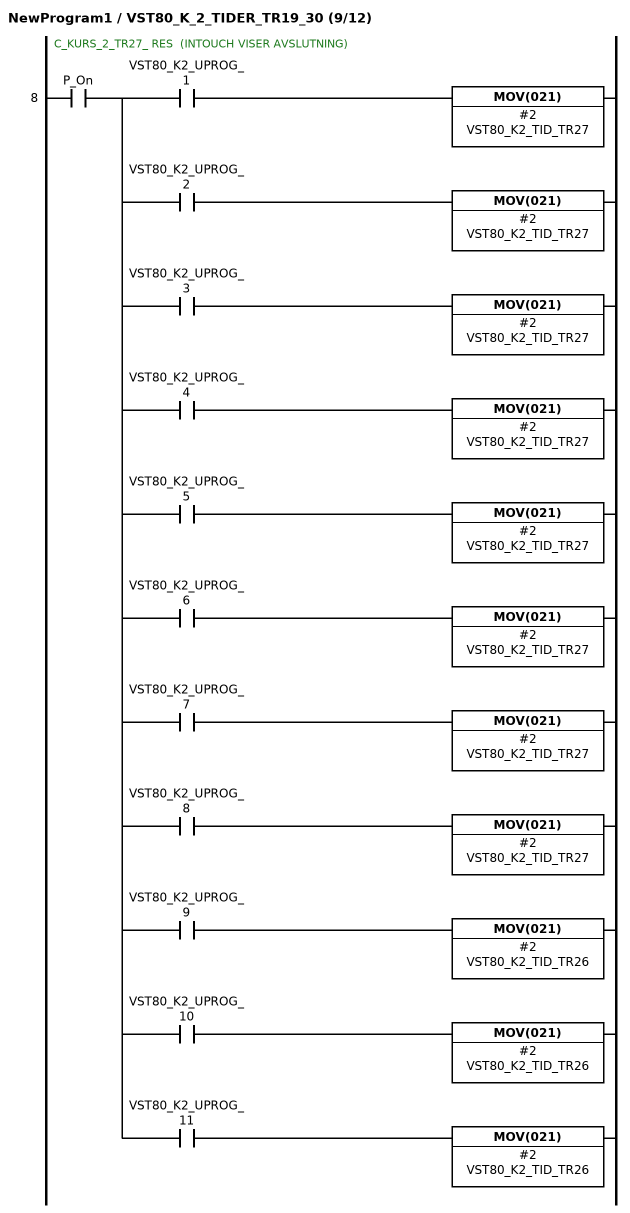
; [picture p192: NewProgram1 / VST80_K_2_TIDER_TR19_30, rungs 8-8]
; rung 8: C_KURS_2_TR27_ RES  (INTOUCH VISER AVSLUTNING)
LD P_On
OUT TR0
AND VST80_K2_UPROG_1
MOV(021) #2 VST80_K2_TID_TR27
LD TR0
AND VST80_K2_UPROG_2
MOV(021) #2 VST80_K2_TID_TR27
LD TR0
AND VST80_K2_UPROG_3
MOV(021) #2 VST80_K2_TID_TR27
LD TR0
AND VST80_K2_UPROG_4
MOV(021) #2 VST80_K2_TID_TR27
LD TR0
AND VST80_K2_UPROG_5
MOV(021) #2 VST80_K2_TID_TR27
LD TR0
AND VST80_K2_UPROG_6
MOV(021) #2 VST80_K2_TID_TR27
LD TR0
AND VST80_K2_UPROG_7
MOV(021) #2 VST80_K2_TID_TR27
LD TR0
AND VST80_K2_UPROG_8
MOV(021) #2 VST80_K2_TID_TR27
LD TR0
AND VST80_K2_UPROG_9
MOV(021) #2 VST80_K2_TID_TR26
LD TR0
AND VST80_K2_UPROG_10
MOV(021) #2 VST80_K2_TID_TR26
LD TR0
AND VST80_K2_UPROG_11
MOV(021) #2 VST80_K2_TID_TR26

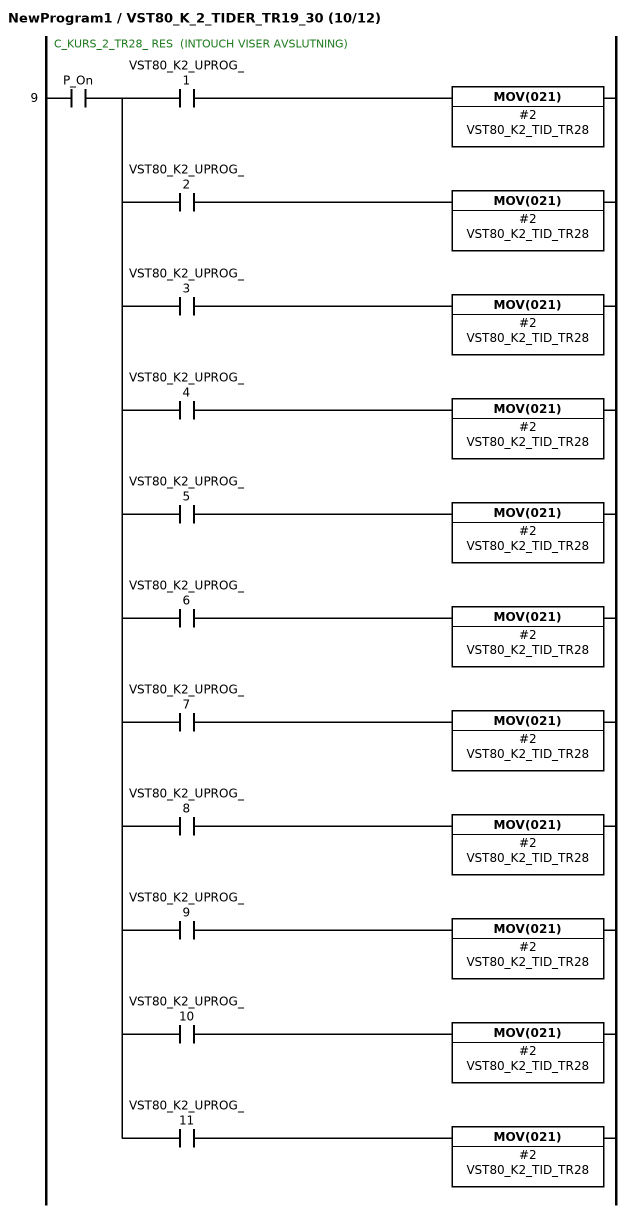
; rung 9: C_KURS_2_TR28_ RES  (INTOUCH VISER AVSLUTNING)
LD P_On
OUT TR0
AND VST80_K2_UPROG_1
MOV(021) #2 VST80_K2_TID_TR28
LD TR0
AND VST80_K2_UPROG_2
MOV(021) #2 VST80_K2_TID_TR28
LD TR0
AND VST80_K2_UPROG_3
MOV(021) #2 VST80_K2_TID_TR28
LD TR0
AND VST80_K2_UPROG_4
MOV(021) #2 VST80_K2_TID_TR28
LD TR0
AND VST80_K2_UPROG_5
MOV(021) #2 VST80_K2_TID_TR28
LD TR0
AND VST80_K2_UPROG_6
MOV(021) #2 VST80_K2_TID_TR28
LD TR0
AND VST80_K2_UPROG_7
MOV(021) #2 VST80_K2_TID_TR28
LD TR0
AND VST80_K2_UPROG_8
MOV(021) #2 VST80_K2_TID_TR28
LD TR0
AND VST80_K2_UPROG_9
MOV(021) #2 VST80_K2_TID_TR28
LD TR0
AND VST80_K2_UPROG_10
MOV(021) #2 VST80_K2_TID_TR28
LD TR0
AND VST80_K2_UPROG_11
MOV(021) #2 VST80_K2_TID_TR28

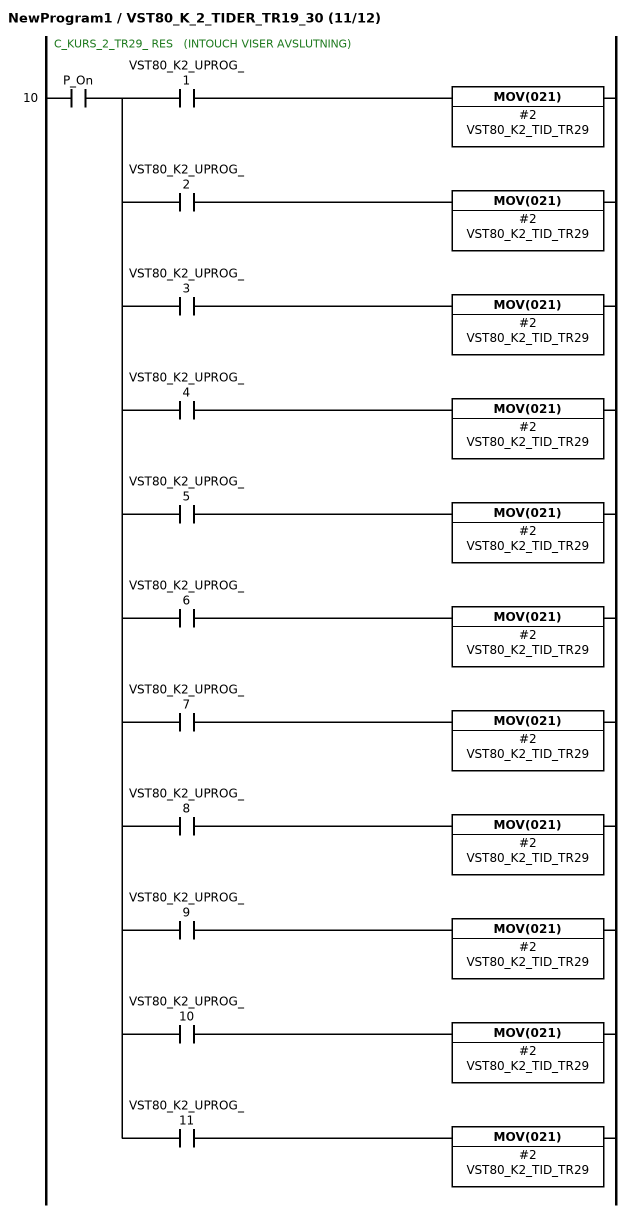
; rung 10: C_KURS_2_TR29_ RES   (INTOUCH VISER AVSLUTNING)
LD P_On
OUT TR0
AND VST80_K2_UPROG_1
MOV(021) #2 VST80_K2_TID_TR29
LD TR0
AND VST80_K2_UPROG_2
MOV(021) #2 VST80_K2_TID_TR29
LD TR0
AND VST80_K2_UPROG_3
MOV(021) #2 VST80_K2_TID_TR29
LD TR0
AND VST80_K2_UPROG_4
MOV(021) #2 VST80_K2_TID_TR29
LD TR0
AND VST80_K2_UPROG_5
MOV(021) #2 VST80_K2_TID_TR29
LD TR0
AND VST80_K2_UPROG_6
MOV(021) #2 VST80_K2_TID_TR29
LD TR0
AND VST80_K2_UPROG_7
MOV(021) #2 VST80_K2_TID_TR29
LD TR0
AND VST80_K2_UPROG_8
MOV(021) #2 VST80_K2_TID_TR29
LD TR0
AND VST80_K2_UPROG_9
MOV(021) #2 VST80_K2_TID_TR29
LD TR0
AND VST80_K2_UPROG_10
MOV(021) #2 VST80_K2_TID_TR29
LD TR0
AND VST80_K2_UPROG_11
MOV(021) #2 VST80_K2_TID_TR29

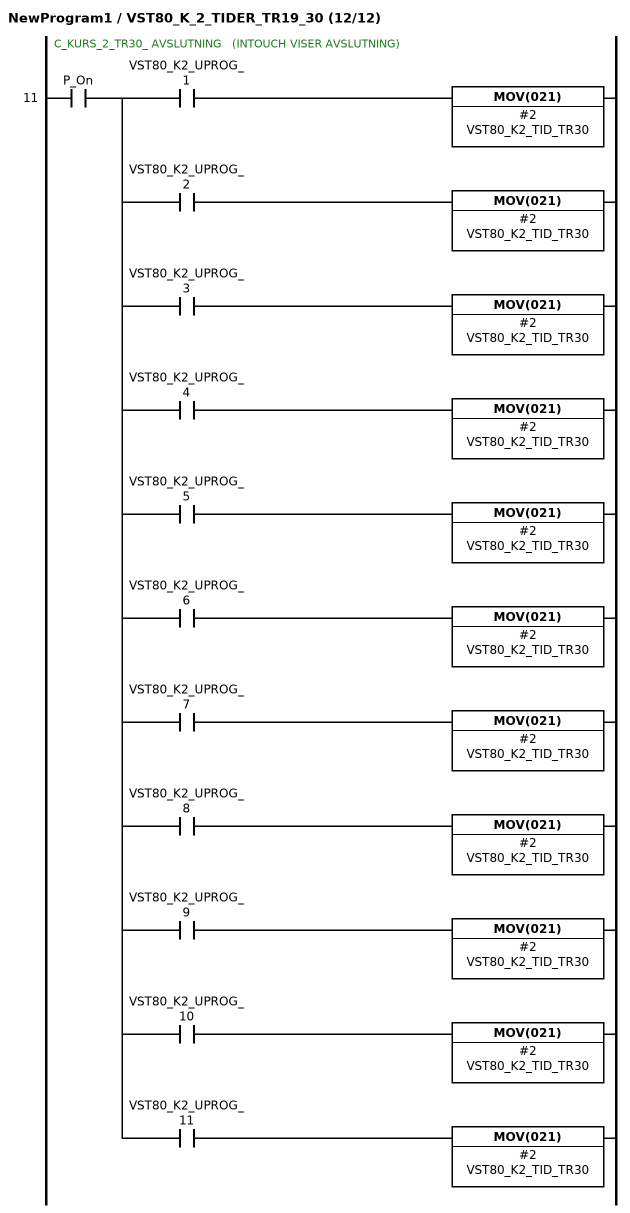
; rung 11: C_KURS_2_TR30_ AVSLUTNING   (INTOUCH VISER AVSLUTNING)
LD P_On
OUT TR0
AND VST80_K2_UPROG_1
MOV(021) #2 VST80_K2_TID_TR30
LD TR0
AND VST80_K2_UPROG_2
MOV(021) #2 VST80_K2_TID_TR30
LD TR0
AND VST80_K2_UPROG_3
MOV(021) #2 VST80_K2_TID_TR30
LD TR0
AND VST80_K2_UPROG_4
MOV(021) #2 VST80_K2_TID_TR30
LD TR0
AND VST80_K2_UPROG_5
MOV(021) #2 VST80_K2_TID_TR30
LD TR0
AND VST80_K2_UPROG_6
MOV(021) #2 VST80_K2_TID_TR30
LD TR0
AND VST80_K2_UPROG_7
MOV(021) #2 VST80_K2_TID_TR30
LD TR0
AND VST80_K2_UPROG_8
MOV(021) #2 VST80_K2_TID_TR30
LD TR0
AND VST80_K2_UPROG_9
MOV(021) #2 VST80_K2_TID_TR30
LD TR0
AND VST80_K2_UPROG_10
MOV(021) #2 VST80_K2_TID_TR30
LD TR0
AND VST80_K2_UPROG_11
MOV(021) #2 VST80_K2_TID_TR30

### Section VST80_K2_TRINN
; Vaskeprogrammet består av 30. hovedtrinn. / Funksjonsbenstabell: 975100-BL48

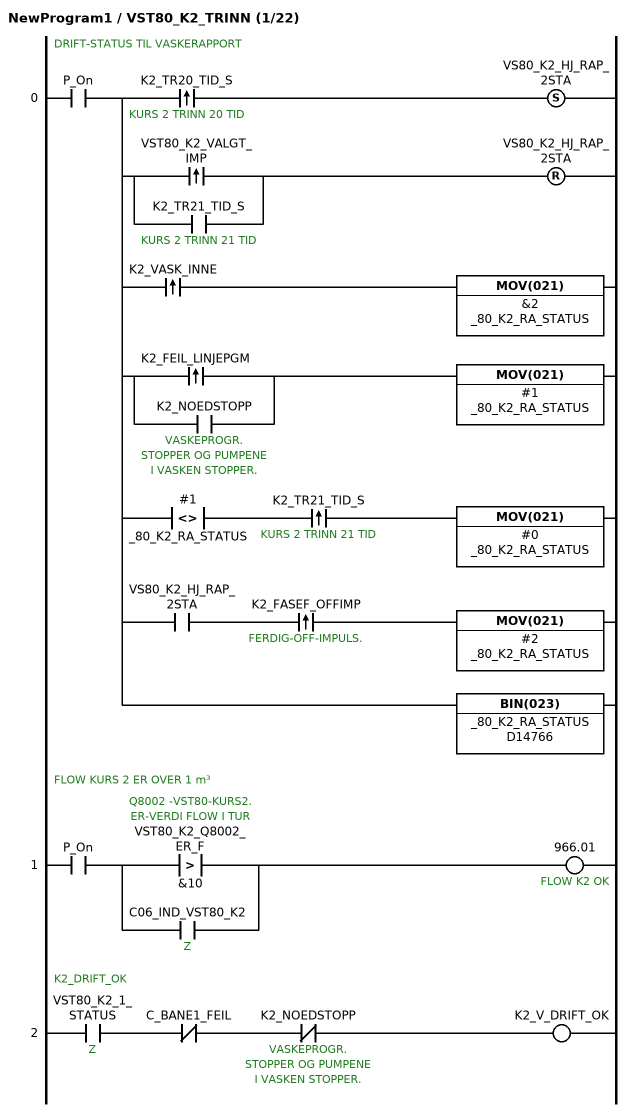
; rung 0: DRIFT-STATUS TIL VASKERAPPORT
LD P_On
OUT TR0
@AND K2_TR20_TID_S  ; KURS 2 TRINN 20 TID
SET VS80_K2_HJ_RAP_2STA
LD TR0
@LD VST80_K2_VALGT_IMP
OR K2_TR21_TID_S  ; KURS 2 TRINN 21 TID
ANDLD
RSET VS80_K2_HJ_RAP_2STA
LD TR0
@AND K2_VASK_INNE
MOV(021) &2 _80_K2_RA_STATUS
LD TR0
@LD K2_FEIL_LINJEPGM
OR K2_NOEDSTOPP  ; VASKEPROGR. STOPPER OG PUMPENE I VASKEN STOPPER.
ANDLD
MOV(021) #1 _80_K2_RA_STATUS
LD TR0
AND<>(305) #1 _80_K2_RA_STATUS
@AND K2_TR21_TID_S  ; KURS 2 TRINN 21 TID
MOV(021) #0 _80_K2_RA_STATUS
LD TR0
AND VS80_K2_HJ_RAP_2STA
@AND K2_FASEF_OFFIMP  ; FERDIG-OFF-IMPULS.
MOV(021) #2 _80_K2_RA_STATUS
LD TR0
BIN(023) _80_K2_RA_STATUS D14766
; rung 1: FLOW KURS 2 ER OVER 1 m³
LD P_On
LD>(320) VST80_K2_Q8002_ER_F &10  ; Q8002 -VST80-KURS2. ER-VERDI FLOW I TUR
OR C06_IND_VST80_K2  ; Z
ANDLD
OUT 966.01  ; FLOW K2 OK
; rung 2: K2_DRIFT_OK
LD VST80_K2_1_STATUS  ; Z
ANDNOT C_BANE1_FEIL
ANDNOT K2_NOEDSTOPP  ; VASKEPROGR. STOPPER OG PUMPENE I VASKEN STOPPER.
OUT K2_V_DRIFT_OK

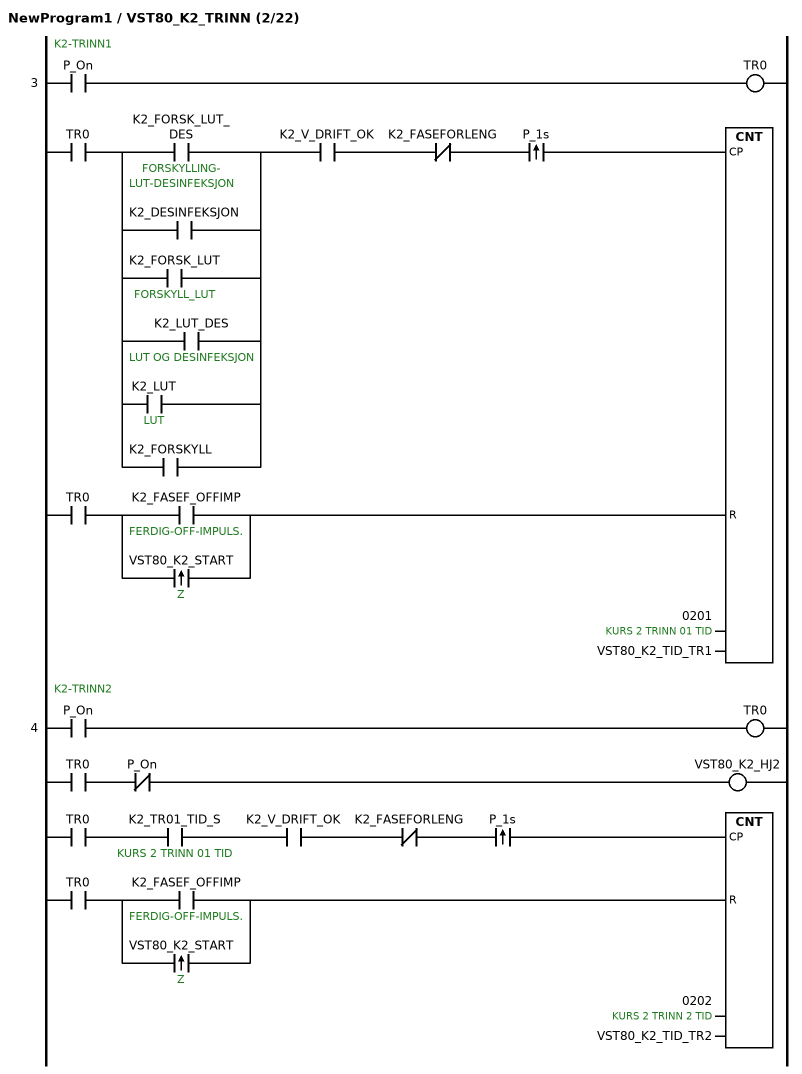
; rung 3: K2-TRINN1
LD P_On
OUT TR0
LD K2_FORSK_LUT_DES  ; FORSKYLLING- LUT-DESINFEKSJON
OR K2_DESINFEKSJON
OR K2_FORSK_LUT  ; FORSKYLL_LUT
OR K2_LUT_DES  ; LUT OG DESINFEKSJON
OR K2_LUT  ; LUT
OR K2_FORSKYLL
ANDLD
AND K2_V_DRIFT_OK
ANDNOT K2_FASEFORLENG
@AND P_1s
LD TR0
LD K2_FASEF_OFFIMP  ; FERDIG-OFF-IMPULS.
@OR VST80_K2_START  ; Z
ANDLD
CNT 0201 VST80_K2_TID_TR1  ; KURS 2 TRINN 01 TID
; rung 4: K2-TRINN2
LD P_On
OUT TR0
ANDNOT P_On
OUT VST80_K2_HJ2
LD TR0
AND K2_TR01_TID_S  ; KURS 2 TRINN 01 TID
AND K2_V_DRIFT_OK
ANDNOT K2_FASEFORLENG
@AND P_1s
LD TR0
LD K2_FASEF_OFFIMP  ; FERDIG-OFF-IMPULS.
@OR VST80_K2_START  ; Z
ANDLD
CNT 0202 VST80_K2_TID_TR2  ; KURS 2 TRINN 2 TID

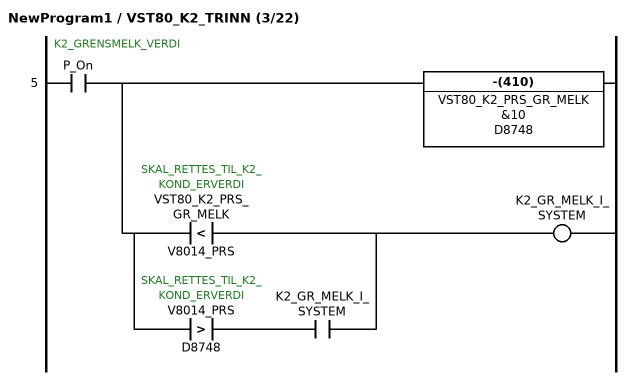
; rung 5: K2_GRENSMELK_VERDI
LD P_On
-(410) VST80_K2_PRS_GR_MELK &10 D8748
LD<(310) VST80_K2_PRS_GR_MELK V8014_PRS  ; SKAL_RETTES_TIL_K2_KOND_ERVERDI
LD>(320) V8014_PRS D8748  ; SKAL_RETTES_TIL_K2_KOND_ERVERDI
AND K2_GR_MELK_I_SYSTEM
ORLD
ANDLD
OUT K2_GR_MELK_I_SYSTEM

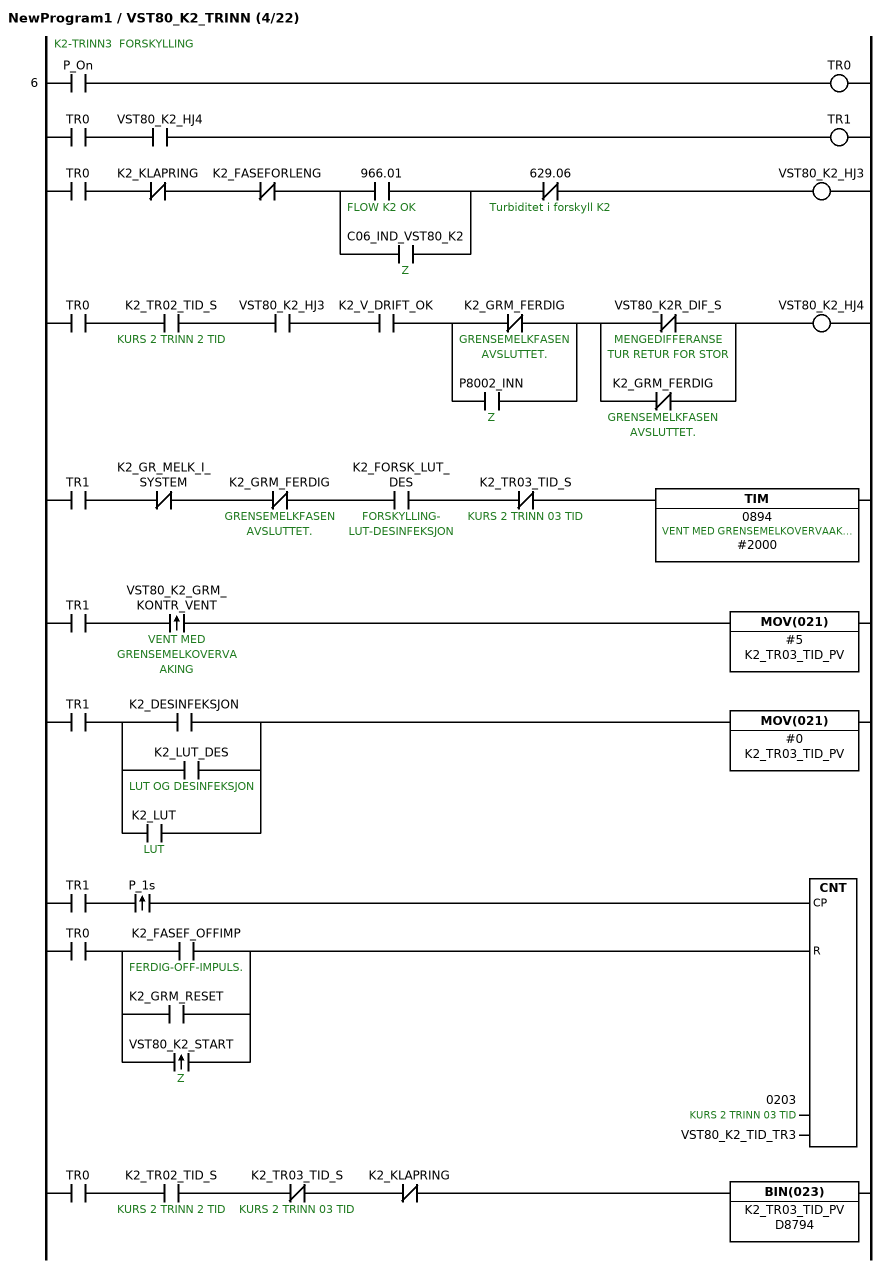
; rung 6: K2-TRINN3  FORSKYLLING
LD P_On
OUT TR0
ANDNOT K2_KLAPRING
ANDNOT K2_FASEFORLENG
LD 966.01  ; FLOW K2 OK
OR C06_IND_VST80_K2  ; Z
ANDLD
ANDNOT 629.06  ; Turbiditet i forskyll K2
OUT VST80_K2_HJ3
LD TR0
AND K2_TR02_TID_S  ; KURS 2 TRINN 2 TID
AND VST80_K2_HJ3
AND K2_V_DRIFT_OK
LDNOT K2_GRM_FERDIG  ; GRENSEMELKFASEN AVSLUTTET.
OR P8002_INN  ; Z
ANDLD
LDNOT VST80_K2R_DIF_S  ; MENGEDIFFERANSE TUR RETUR FOR STOR
ORNOT K2_GRM_FERDIG  ; GRENSEMELKFASEN AVSLUTTET.
ANDLD
OUT VST80_K2_HJ4
LD TR0
AND VST80_K2_HJ4
OUT TR1
ANDNOT K2_GR_MELK_I_SYSTEM
ANDNOT K2_GRM_FERDIG  ; GRENSEMELKFASEN AVSLUTTET.
AND K2_FORSK_LUT_DES  ; FORSKYLLING- LUT-DESINFEKSJON
ANDNOT K2_TR03_TID_S  ; KURS 2 TRINN 03 TID
TIM 0894 #2000  ; VENT MED GRENSEMELKOVERVAAKING
LD TR1
@AND VST80_K2_GRM_KONTR_VENT  ; VENT MED GRENSEMELKOVERVAAKING
MOV(021) #5 K2_TR03_TID_PV
LD TR1
LD K2_DESINFEKSJON
OR K2_LUT_DES  ; LUT OG DESINFEKSJON
OR K2_LUT  ; LUT
ANDLD
MOV(021) #0 K2_TR03_TID_PV
LD TR1
@AND P_1s
LD TR0
LD K2_FASEF_OFFIMP  ; FERDIG-OFF-IMPULS.
OR K2_GRM_RESET
@OR VST80_K2_START  ; Z
ANDLD
CNT 0203 VST80_K2_TID_TR3  ; KURS 2 TRINN 03 TID
LD TR0
AND K2_TR02_TID_S  ; KURS 2 TRINN 2 TID
ANDNOT K2_TR03_TID_S  ; KURS 2 TRINN 03 TID
ANDNOT K2_KLAPRING
BIN(023) K2_TR03_TID_PV D8794

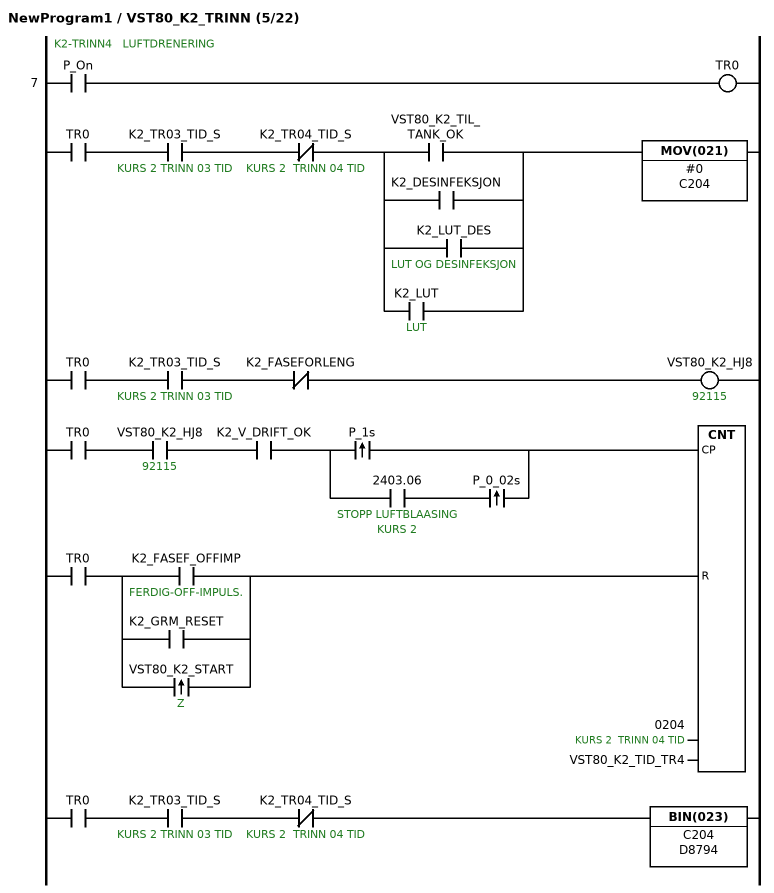
; rung 7: K2-TRINN4   LUFTDRENERING
LD P_On
OUT TR0
AND K2_TR03_TID_S  ; KURS 2 TRINN 03 TID
ANDNOT K2_TR04_TID_S  ; KURS 2  TRINN 04 TID
LD VST80_K2_TIL_TANK_OK
OR K2_DESINFEKSJON
OR K2_LUT_DES  ; LUT OG DESINFEKSJON
OR K2_LUT  ; LUT
ANDLD
MOV(021) #0 C204
LD TR0
AND K2_TR03_TID_S  ; KURS 2 TRINN 03 TID
ANDNOT K2_FASEFORLENG
OUT VST80_K2_HJ8  ; 92115
LD TR0
AND VST80_K2_HJ8  ; 92115
AND K2_V_DRIFT_OK
@LD P_1s
LD 2403.06  ; STOPP LUFTBLAASING KURS 2
@AND P_0_02s
ORLD
ANDLD
LD TR0
LD K2_FASEF_OFFIMP  ; FERDIG-OFF-IMPULS.
OR K2_GRM_RESET
@OR VST80_K2_START  ; Z
ANDLD
CNT 0204 VST80_K2_TID_TR4  ; KURS 2  TRINN 04 TID
LD TR0
AND K2_TR03_TID_S  ; KURS 2 TRINN 03 TID
ANDNOT K2_TR04_TID_S  ; KURS 2  TRINN 04 TID
BIN(023) C204 D8794

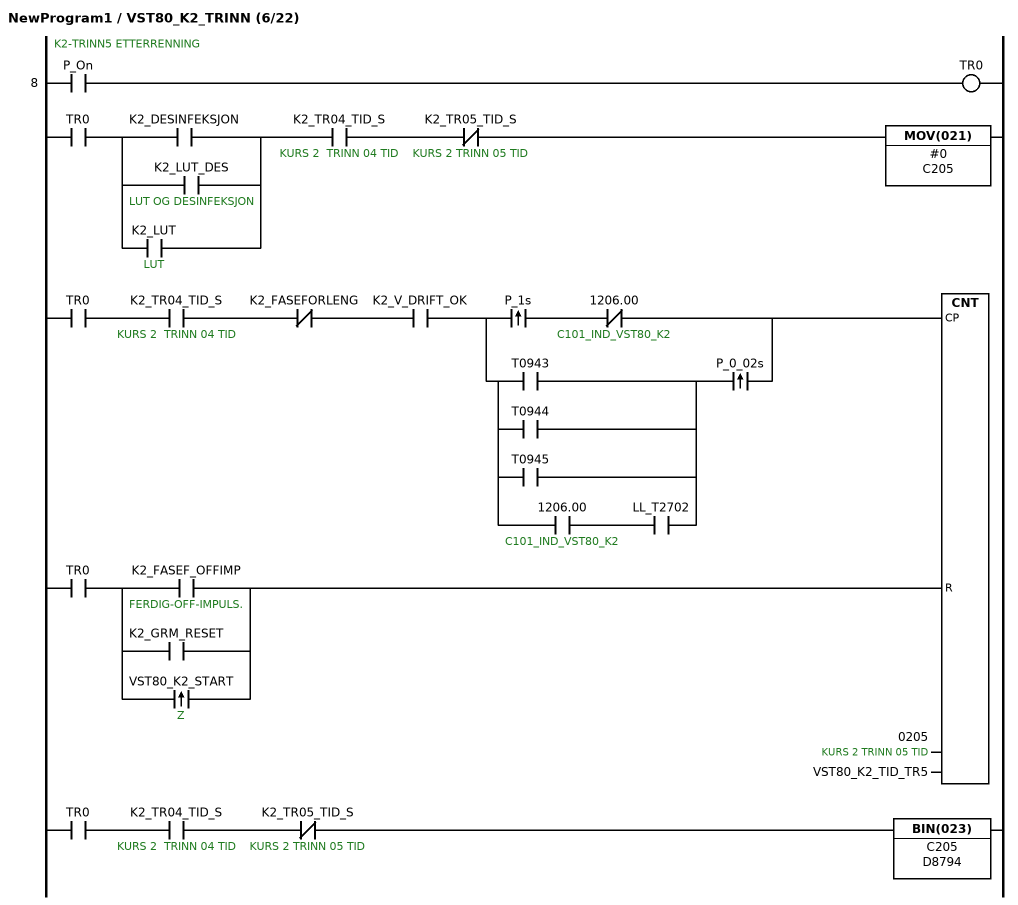
; rung 8: K2-TRINN5 ETTERRENNING
LD P_On
OUT TR0
LD K2_DESINFEKSJON
OR K2_LUT_DES  ; LUT OG DESINFEKSJON
OR K2_LUT  ; LUT
ANDLD
AND K2_TR04_TID_S  ; KURS 2  TRINN 04 TID
ANDNOT K2_TR05_TID_S  ; KURS 2 TRINN 05 TID
MOV(021) #0 C205
LD TR0
AND K2_TR04_TID_S  ; KURS 2  TRINN 04 TID
ANDNOT K2_FASEFORLENG
AND K2_V_DRIFT_OK
@LD P_1s
ANDNOT 1206.00  ; C101_IND_VST80_K2
LD T0943
OR T0944
OR T0945
LD 1206.00  ; C101_IND_VST80_K2
AND LL_T2702
ORLD
@AND P_0_02s
ORLD
ANDLD
LD TR0
LD K2_FASEF_OFFIMP  ; FERDIG-OFF-IMPULS.
OR K2_GRM_RESET
@OR VST80_K2_START  ; Z
ANDLD
CNT 0205 VST80_K2_TID_TR5  ; KURS 2 TRINN 05 TID
LD TR0
AND K2_TR04_TID_S  ; KURS 2  TRINN 04 TID
ANDNOT K2_TR05_TID_S  ; KURS 2 TRINN 05 TID
BIN(023) C205 D8794

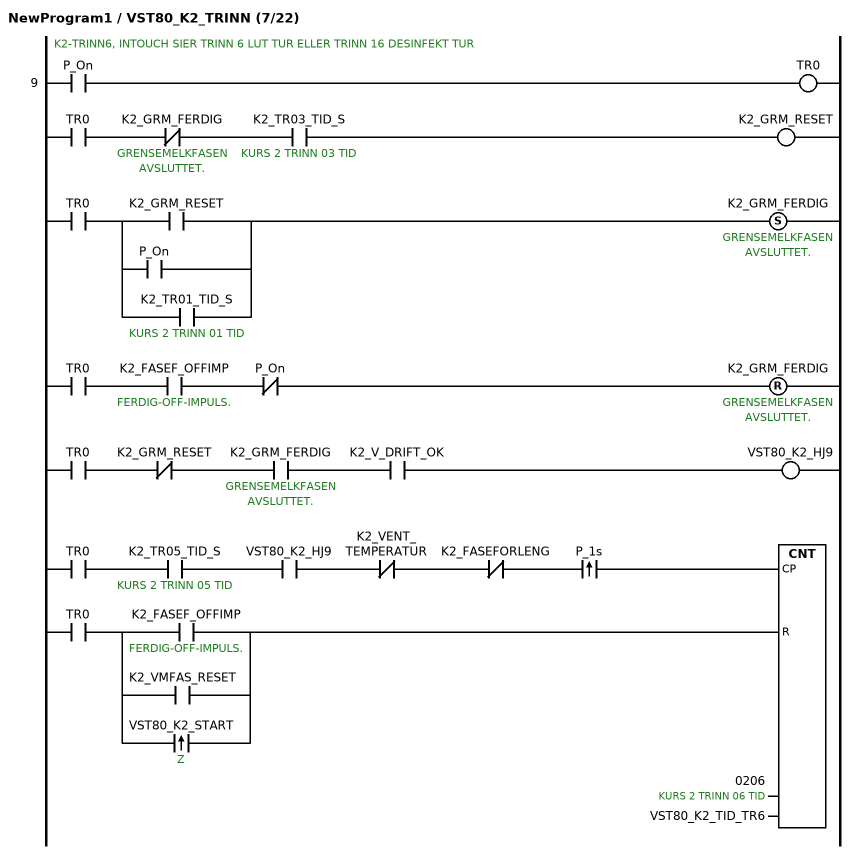
; rung 9: K2-TRINN6, INTOUCH SIER TRINN 6 LUT TUR ELLER TRINN 16 DESINFEKT TUR
LD P_On
OUT TR0
ANDNOT K2_GRM_FERDIG  ; GRENSEMELKFASEN AVSLUTTET.
AND K2_TR03_TID_S  ; KURS 2 TRINN 03 TID
OUT K2_GRM_RESET
LD TR0
LD K2_GRM_RESET
OR P_On
OR K2_TR01_TID_S  ; KURS 2 TRINN 01 TID
ANDLD
SET K2_GRM_FERDIG  ; GRENSEMELKFASEN AVSLUTTET.
LD TR0
AND K2_FASEF_OFFIMP  ; FERDIG-OFF-IMPULS.
ANDNOT P_On
RSET K2_GRM_FERDIG  ; GRENSEMELKFASEN AVSLUTTET.
LD TR0
ANDNOT K2_GRM_RESET
AND K2_GRM_FERDIG  ; GRENSEMELKFASEN AVSLUTTET.
AND K2_V_DRIFT_OK
OUT VST80_K2_HJ9
LD TR0
AND K2_TR05_TID_S  ; KURS 2 TRINN 05 TID
AND VST80_K2_HJ9
ANDNOT K2_VENT_TEMPERATUR
ANDNOT K2_FASEFORLENG
@AND P_1s
LD TR0
LD K2_FASEF_OFFIMP  ; FERDIG-OFF-IMPULS.
OR K2_VMFAS_RESET
@OR VST80_K2_START  ; Z
ANDLD
CNT 0206 VST80_K2_TID_TR6  ; KURS 2 TRINN 06 TID

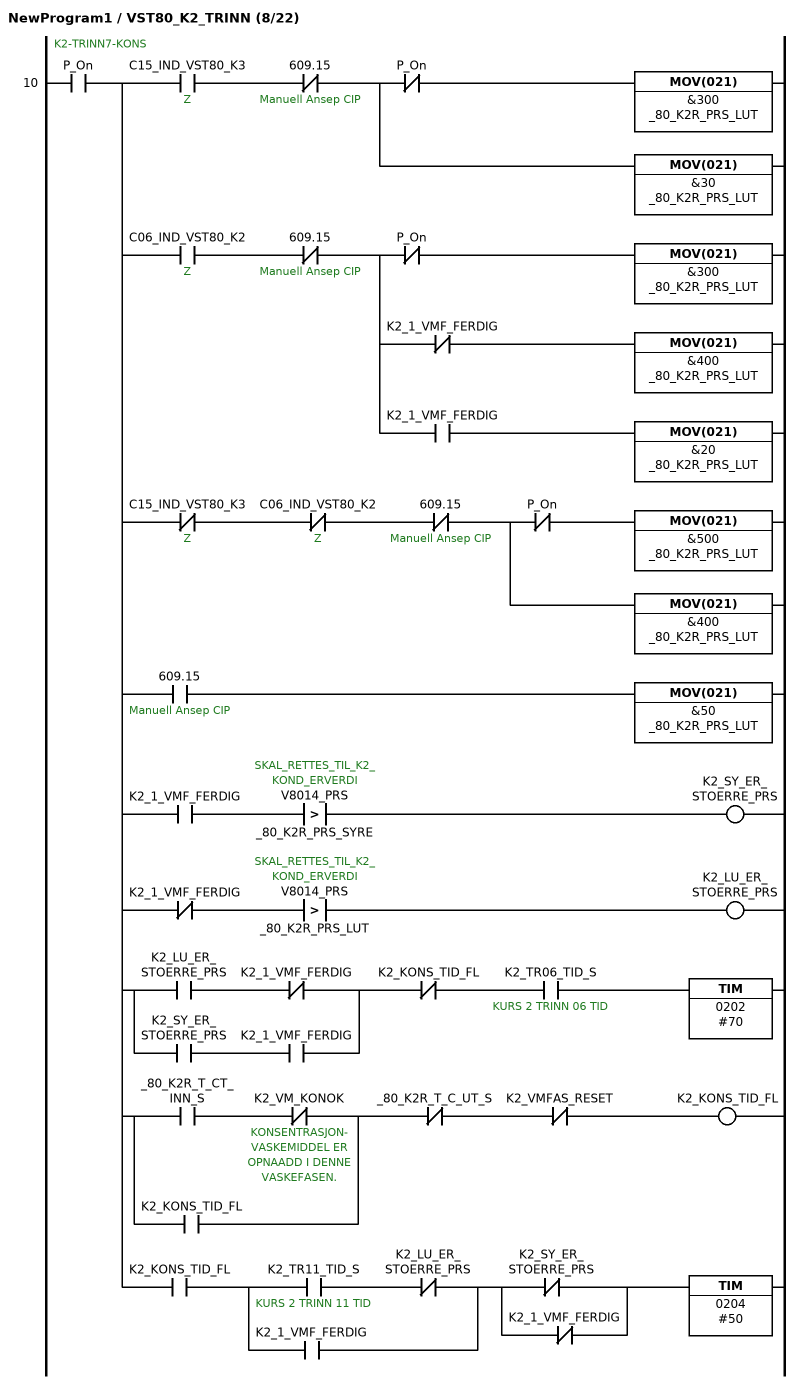
; rung 10: K2-TRINN7-KONS
LD P_On
OUT TR0
AND C15_IND_VST80_K3  ; Z
ANDNOT 609.15  ; Manuell Ansep CIP
OUT TR1
ANDNOT P_On
MOV(021) &300 _80_K2R_PRS_LUT
LD TR1
MOV(021) &30 _80_K2R_PRS_LUT
LD TR0
AND C06_IND_VST80_K2  ; Z
ANDNOT 609.15  ; Manuell Ansep CIP
OUT TR1
ANDNOT P_On
MOV(021) &300 _80_K2R_PRS_LUT
LD TR1
ANDNOT K2_1_VMF_FERDIG
MOV(021) &400 _80_K2R_PRS_LUT
LD TR1
AND K2_1_VMF_FERDIG
MOV(021) &20 _80_K2R_PRS_LUT
LD TR0
ANDNOT C15_IND_VST80_K3  ; Z
ANDNOT C06_IND_VST80_K2  ; Z
ANDNOT 609.15  ; Manuell Ansep CIP
OUT TR1
ANDNOT P_On
MOV(021) &500 _80_K2R_PRS_LUT
LD TR1
MOV(021) &400 _80_K2R_PRS_LUT
LD TR0
AND 609.15  ; Manuell Ansep CIP
MOV(021) &50 _80_K2R_PRS_LUT
LD TR0
AND K2_1_VMF_FERDIG
AND>(320) V8014_PRS _80_K2R_PRS_SYRE  ; SKAL_RETTES_TIL_K2_KOND_ERVERDI
OUT K2_SY_ER_STOERRE_PRS
LD TR0
ANDNOT K2_1_VMF_FERDIG
AND>(320) V8014_PRS _80_K2R_PRS_LUT  ; SKAL_RETTES_TIL_K2_KOND_ERVERDI
OUT K2_LU_ER_STOERRE_PRS
LD TR0
LD K2_LU_ER_STOERRE_PRS
ANDNOT K2_1_VMF_FERDIG
LD K2_SY_ER_STOERRE_PRS
AND K2_1_VMF_FERDIG
ORLD
ANDLD
ANDNOT K2_KONS_TID_FL
AND K2_TR06_TID_S  ; KURS 2 TRINN 06 TID
TIM 0202 #70
LD TR0
LD _80_K2R_T_CT_INN_S
ANDNOT K2_VM_KONOK  ; KONSENTRASJON-VASKEMIDDEL ER OPNAADD I DENNE VASKEFASEN.
OR K2_KONS_TID_FL
ANDLD
ANDNOT _80_K2R_T_C_UT_S
ANDNOT K2_VMFAS_RESET
OUT K2_KONS_TID_FL
LD TR0
AND K2_KONS_TID_FL
LD K2_TR11_TID_S  ; KURS 2 TRINN 11 TID
ANDNOT K2_LU_ER_STOERRE_PRS
OR K2_1_VMF_FERDIG
ANDLD
LDNOT K2_SY_ER_STOERRE_PRS
ORNOT K2_1_VMF_FERDIG
ANDLD
TIM 0204 #50

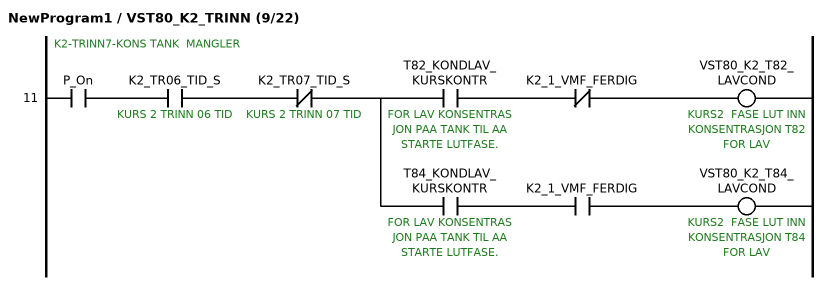
; rung 11: K2-TRINN7-KONS TANK  MANGLER
LD P_On
AND K2_TR06_TID_S  ; KURS 2 TRINN 06 TID
ANDNOT K2_TR07_TID_S  ; KURS 2 TRINN 07 TID
OUT TR0
AND T82_KONDLAV_KURSKONTR  ; FOR LAV KONSENTRASJON PAA TANK TIL AA STARTE LUTFASE.
ANDNOT K2_1_VMF_FERDIG
OUT VST80_K2_T82_LAVCOND  ; KURS2  FASE LUT INN KONSENTRASJON T82 FOR LAV
LD TR0
AND T84_KONDLAV_KURSKONTR  ; FOR LAV KONSENTRASJON PAA TANK TIL AA STARTE LUTFASE.
AND K2_1_VMF_FERDIG
OUT VST80_K2_T84_LAVCOND  ; KURS2  FASE LUT INN KONSENTRASJON T84 FOR LAV

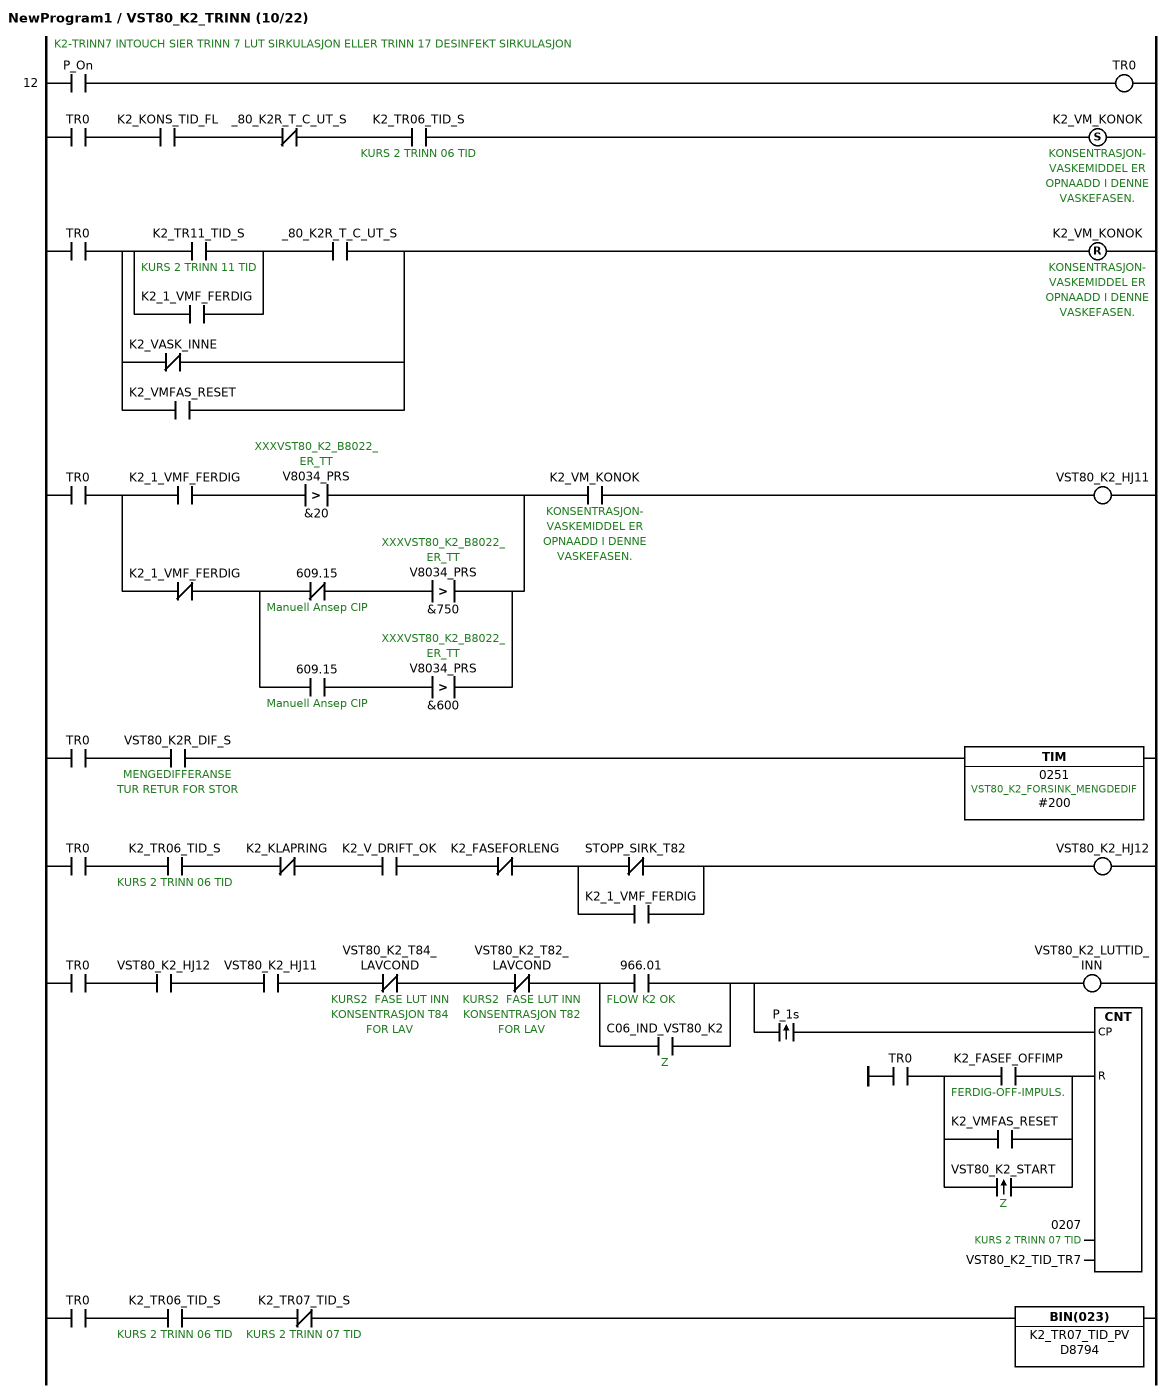
; rung 12: K2-TRINN7 INTOUCH SIER TRINN 7 LUT SIRKULASJON ELLER TRINN 17 DESINFEKT SIRKULASJON
LD P_On
OUT TR0
AND K2_KONS_TID_FL
ANDNOT _80_K2R_T_C_UT_S
AND K2_TR06_TID_S  ; KURS 2 TRINN 06 TID
SET K2_VM_KONOK  ; KONSENTRASJON-VASKEMIDDEL ER OPNAADD I DENNE VASKEFASEN.
LD TR0
LD K2_TR11_TID_S  ; KURS 2 TRINN 11 TID
OR K2_1_VMF_FERDIG
AND _80_K2R_T_C_UT_S
ORNOT K2_VASK_INNE
OR K2_VMFAS_RESET
ANDLD
RSET K2_VM_KONOK  ; KONSENTRASJON-VASKEMIDDEL ER OPNAADD I DENNE VASKEFASEN.
LD TR0
LD K2_1_VMF_FERDIG
AND>(320) V8034_PRS &20  ; XXXVST80_K2_B8022_ER_TT
LDNOT K2_1_VMF_FERDIG
LDNOT 609.15  ; Manuell Ansep CIP
AND>(320) V8034_PRS &750  ; XXXVST80_K2_B8022_ER_TT
LD 609.15  ; Manuell Ansep CIP
AND>(320) V8034_PRS &600  ; XXXVST80_K2_B8022_ER_TT
ORLD
ANDLD
ORLD
ANDLD
AND K2_VM_KONOK  ; KONSENTRASJON-VASKEMIDDEL ER OPNAADD I DENNE VASKEFASEN.
OUT VST80_K2_HJ11
LD TR0
AND VST80_K2R_DIF_S  ; MENGEDIFFERANSE TUR RETUR FOR STOR
TIM 0251 #200  ; VST80_K2_FORSINK_MENGDEDIF
LD TR0
AND K2_TR06_TID_S  ; KURS 2 TRINN 06 TID
ANDNOT K2_KLAPRING
AND K2_V_DRIFT_OK
ANDNOT K2_FASEFORLENG
LDNOT STOPP_SIRK_T82
OR K2_1_VMF_FERDIG
ANDLD
OUT VST80_K2_HJ12
LD TR0
AND VST80_K2_HJ12
AND VST80_K2_HJ11
ANDNOT VST80_K2_T84_LAVCOND  ; KURS2  FASE LUT INN KONSENTRASJON T84 FOR LAV
ANDNOT VST80_K2_T82_LAVCOND  ; KURS2  FASE LUT INN KONSENTRASJON T82 FOR LAV
LD 966.01  ; FLOW K2 OK
OR C06_IND_VST80_K2  ; Z
ANDLD
OUT VST80_K2_LUTTID_INN
@AND P_1s
LD TR0
LD K2_FASEF_OFFIMP  ; FERDIG-OFF-IMPULS.
OR K2_VMFAS_RESET
@OR VST80_K2_START  ; Z
ANDLD
CNT 0207 VST80_K2_TID_TR7  ; KURS 2 TRINN 07 TID
LD TR0
AND K2_TR06_TID_S  ; KURS 2 TRINN 06 TID
ANDNOT K2_TR07_TID_S  ; KURS 2 TRINN 07 TID
BIN(023) K2_TR07_TID_PV D8794

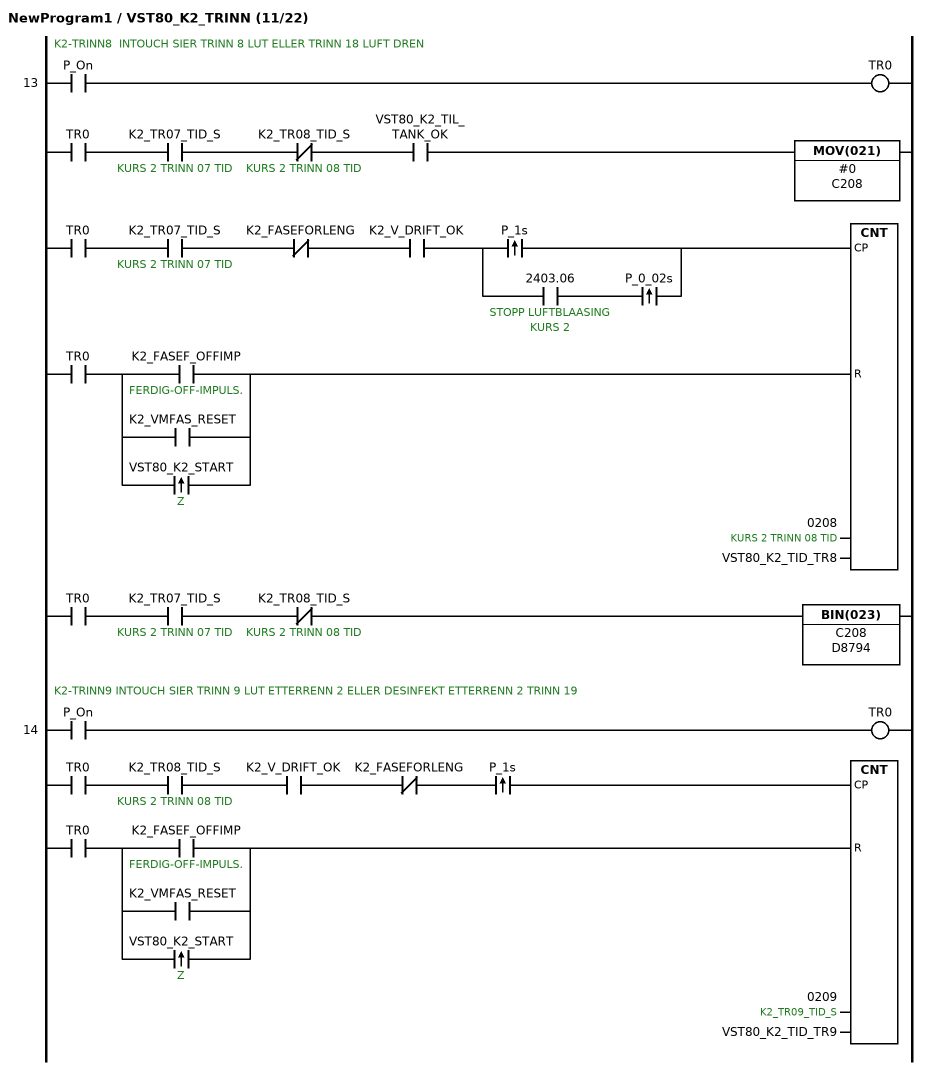
; rung 13: K2-TRINN8  INTOUCH SIER TRINN 8 LUT ELLER TRINN 18 LUFT DREN
LD P_On
OUT TR0
AND K2_TR07_TID_S  ; KURS 2 TRINN 07 TID
ANDNOT K2_TR08_TID_S  ; KURS 2 TRINN 08 TID
AND VST80_K2_TIL_TANK_OK
MOV(021) #0 C208
LD TR0
AND K2_TR07_TID_S  ; KURS 2 TRINN 07 TID
ANDNOT K2_FASEFORLENG
AND K2_V_DRIFT_OK
@LD P_1s
LD 2403.06  ; STOPP LUFTBLAASING KURS 2
@AND P_0_02s
ORLD
ANDLD
LD TR0
LD K2_FASEF_OFFIMP  ; FERDIG-OFF-IMPULS.
OR K2_VMFAS_RESET
@OR VST80_K2_START  ; Z
ANDLD
CNT 0208 VST80_K2_TID_TR8  ; KURS 2 TRINN 08 TID
LD TR0
AND K2_TR07_TID_S  ; KURS 2 TRINN 07 TID
ANDNOT K2_TR08_TID_S  ; KURS 2 TRINN 08 TID
BIN(023) C208 D8794
; rung 14: K2-TRINN9 INTOUCH SIER TRINN 9 LUT ETTERRENN 2 ELLER DESINFEKT ETTERRENN 2 TRINN 19
LD P_On
OUT TR0
AND K2_TR08_TID_S  ; KURS 2 TRINN 08 TID
AND K2_V_DRIFT_OK
ANDNOT K2_FASEFORLENG
@AND P_1s
LD TR0
LD K2_FASEF_OFFIMP  ; FERDIG-OFF-IMPULS.
OR K2_VMFAS_RESET
@OR VST80_K2_START  ; Z
ANDLD
CNT 0209 VST80_K2_TID_TR9  ; K2_TR09_TID_S

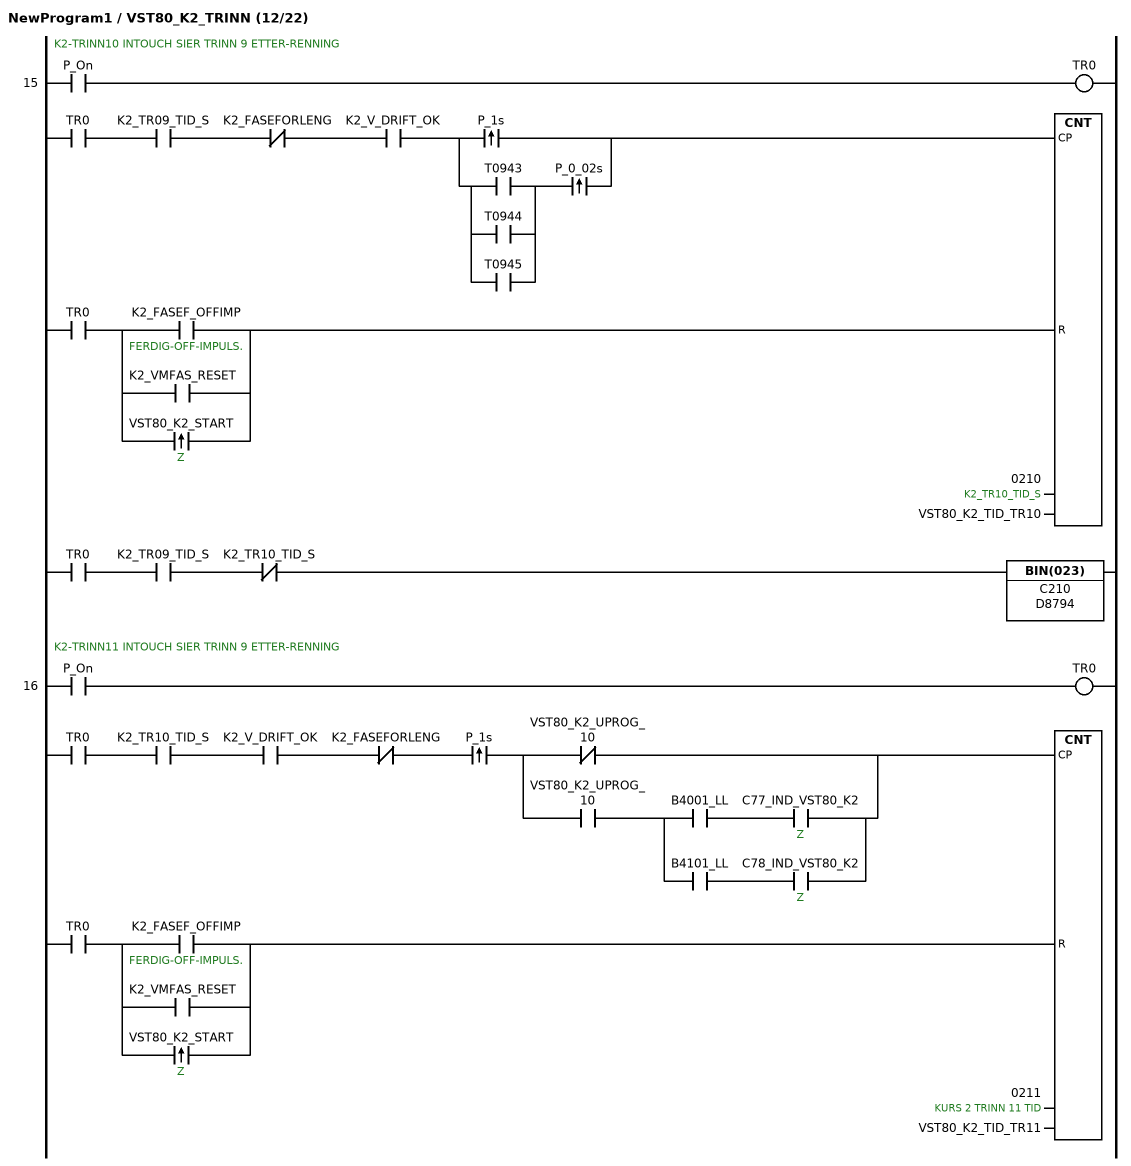
; rung 15: K2-TRINN10 INTOUCH SIER TRINN 9 ETTER-RENNING
LD P_On
OUT TR0
AND K2_TR09_TID_S
ANDNOT K2_FASEFORLENG
AND K2_V_DRIFT_OK
@LD P_1s
LD T0943
OR T0944
OR T0945
@AND P_0_02s
ORLD
ANDLD
LD TR0
LD K2_FASEF_OFFIMP  ; FERDIG-OFF-IMPULS.
OR K2_VMFAS_RESET
@OR VST80_K2_START  ; Z
ANDLD
CNT 0210 VST80_K2_TID_TR10  ; K2_TR10_TID_S
LD TR0
AND K2_TR09_TID_S
ANDNOT K2_TR10_TID_S
BIN(023) C210 D8794
; rung 16: K2-TRINN11 INTOUCH SIER TRINN 9 ETTER-RENNING
LD P_On
OUT TR0
AND K2_TR10_TID_S
AND K2_V_DRIFT_OK
ANDNOT K2_FASEFORLENG
@AND P_1s
LDNOT VST80_K2_UPROG_10
LD VST80_K2_UPROG_10
LD B4001_LL
AND C77_IND_VST80_K2  ; Z
LD B4101_LL
AND C78_IND_VST80_K2  ; Z
ORLD
ANDLD
ORLD
ANDLD
LD TR0
LD K2_FASEF_OFFIMP  ; FERDIG-OFF-IMPULS.
OR K2_VMFAS_RESET
@OR VST80_K2_START  ; Z
ANDLD
CNT 0211 VST80_K2_TID_TR11  ; KURS 2 TRINN 11 TID

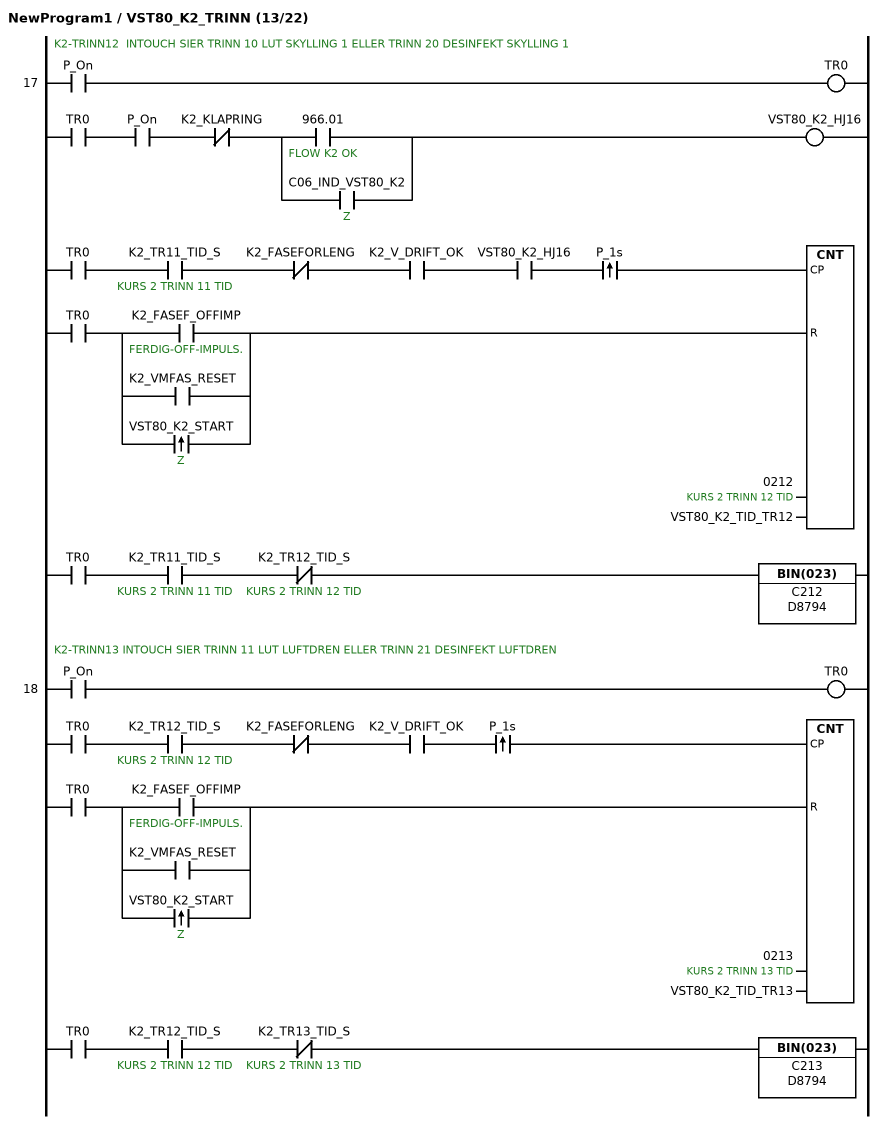
; rung 17: K2-TRINN12  INTOUCH SIER TRINN 10 LUT SKYLLING 1 ELLER TRINN 20 DESINFEKT SKYLLING 1
LD P_On
OUT TR0
AND P_On
ANDNOT K2_KLAPRING
LD 966.01  ; FLOW K2 OK
OR C06_IND_VST80_K2  ; Z
ANDLD
OUT VST80_K2_HJ16
LD TR0
AND K2_TR11_TID_S  ; KURS 2 TRINN 11 TID
ANDNOT K2_FASEFORLENG
AND K2_V_DRIFT_OK
AND VST80_K2_HJ16
@AND P_1s
LD TR0
LD K2_FASEF_OFFIMP  ; FERDIG-OFF-IMPULS.
OR K2_VMFAS_RESET
@OR VST80_K2_START  ; Z
ANDLD
CNT 0212 VST80_K2_TID_TR12  ; KURS 2 TRINN 12 TID
LD TR0
AND K2_TR11_TID_S  ; KURS 2 TRINN 11 TID
ANDNOT K2_TR12_TID_S  ; KURS 2 TRINN 12 TID
BIN(023) C212 D8794
; rung 18: K2-TRINN13 INTOUCH SIER TRINN 11 LUT LUFTDREN ELLER TRINN 21 DESINFEKT LUFTDREN
LD P_On
OUT TR0
AND K2_TR12_TID_S  ; KURS 2 TRINN 12 TID
ANDNOT K2_FASEFORLENG
AND K2_V_DRIFT_OK
@AND P_1s
LD TR0
LD K2_FASEF_OFFIMP  ; FERDIG-OFF-IMPULS.
OR K2_VMFAS_RESET
@OR VST80_K2_START  ; Z
ANDLD
CNT 0213 VST80_K2_TID_TR13  ; KURS 2 TRINN 13 TID
LD TR0
AND K2_TR12_TID_S  ; KURS 2 TRINN 12 TID
ANDNOT K2_TR13_TID_S  ; KURS 2 TRINN 13 TID
BIN(023) C213 D8794

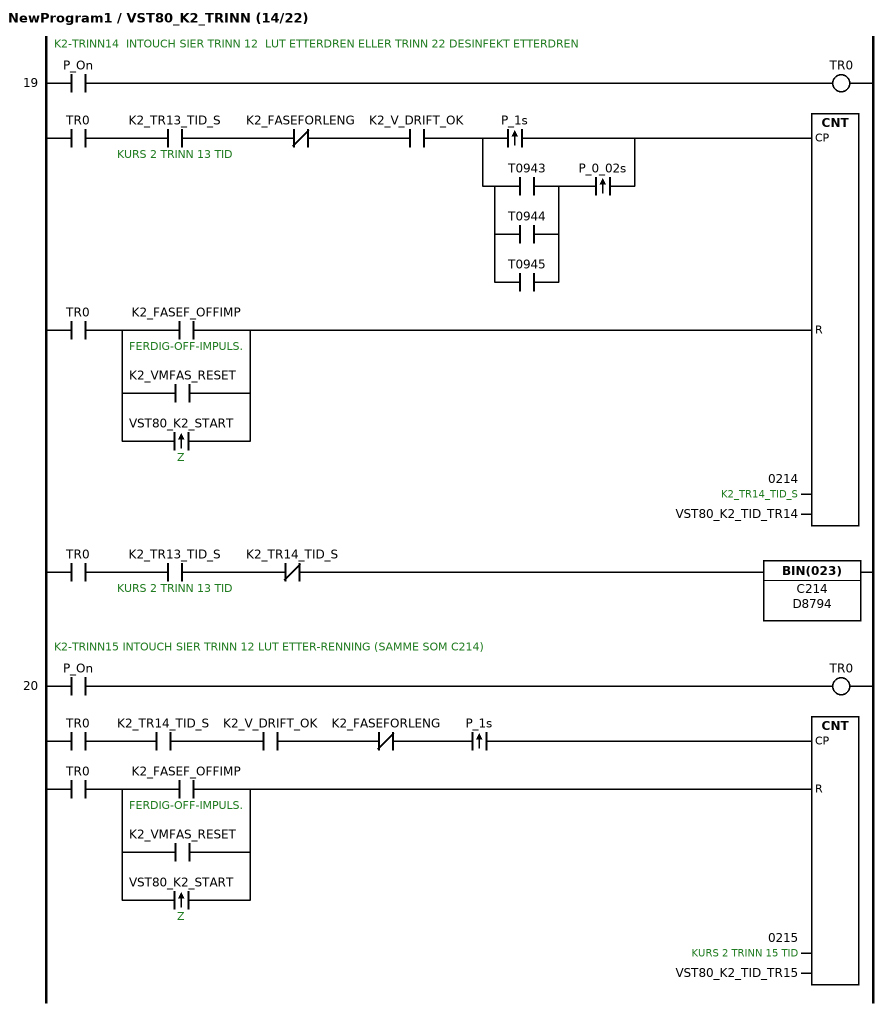
; rung 19: K2-TRINN14  INTOUCH SIER TRINN 12  LUT ETTERDREN ELLER TRINN 22 DESINFEKT ETTERDREN
LD P_On
OUT TR0
AND K2_TR13_TID_S  ; KURS 2 TRINN 13 TID
ANDNOT K2_FASEFORLENG
AND K2_V_DRIFT_OK
@LD P_1s
LD T0943
OR T0944
OR T0945
@AND P_0_02s
ORLD
ANDLD
LD TR0
LD K2_FASEF_OFFIMP  ; FERDIG-OFF-IMPULS.
OR K2_VMFAS_RESET
@OR VST80_K2_START  ; Z
ANDLD
CNT 0214 VST80_K2_TID_TR14  ; K2_TR14_TID_S
LD TR0
AND K2_TR13_TID_S  ; KURS 2 TRINN 13 TID
ANDNOT K2_TR14_TID_S
BIN(023) C214 D8794
; rung 20: K2-TRINN15 INTOUCH SIER TRINN 12 LUT ETTER-RENNING (SAMME SOM C214)
LD P_On
OUT TR0
AND K2_TR14_TID_S
AND K2_V_DRIFT_OK
ANDNOT K2_FASEFORLENG
@AND P_1s
LD TR0
LD K2_FASEF_OFFIMP  ; FERDIG-OFF-IMPULS.
OR K2_VMFAS_RESET
@OR VST80_K2_START  ; Z
ANDLD
CNT 0215 VST80_K2_TID_TR15  ; KURS 2 TRINN 15 TID

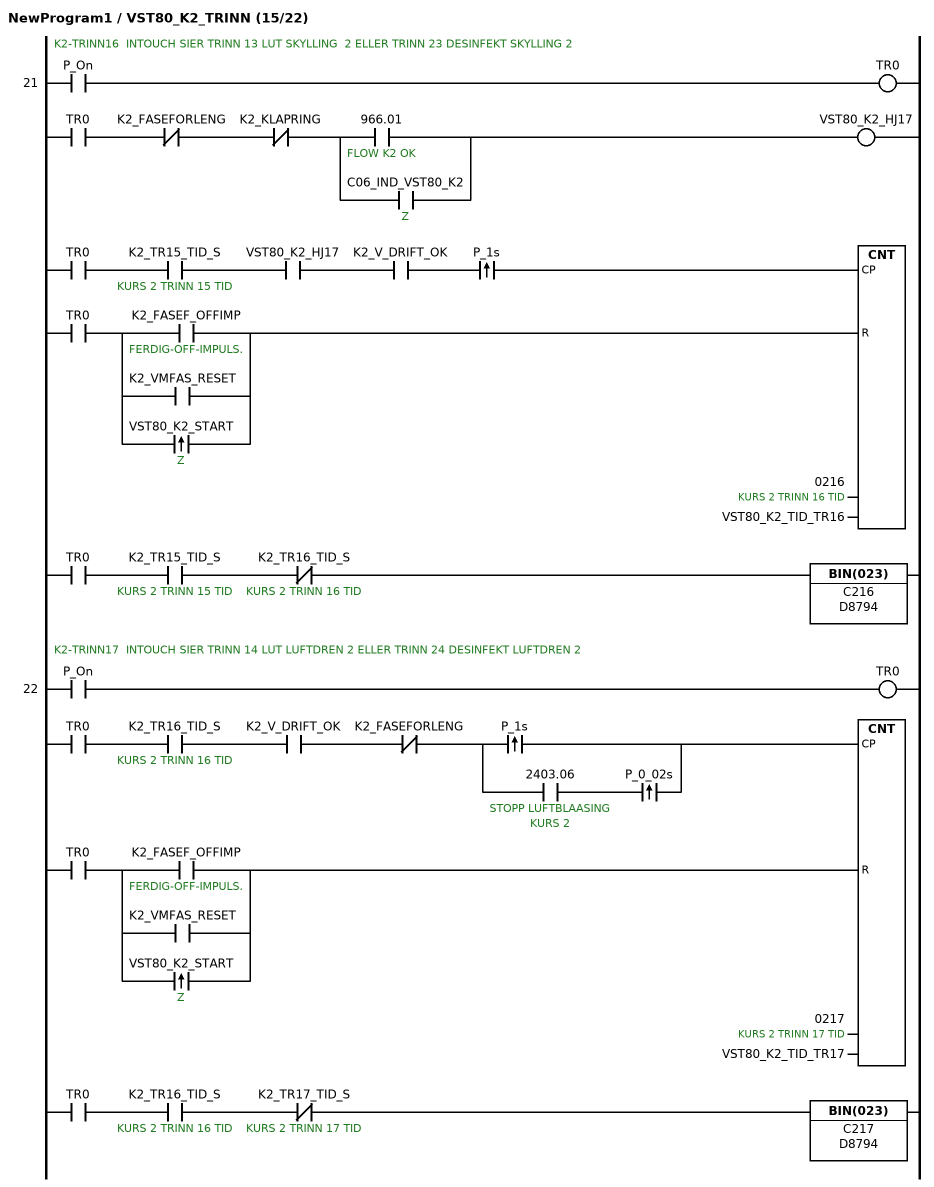
; rung 21: K2-TRINN16  INTOUCH SIER TRINN 13 LUT SKYLLING  2 ELLER TRINN 23 DESINFEKT SKYLLING 2
LD P_On
OUT TR0
ANDNOT K2_FASEFORLENG
ANDNOT K2_KLAPRING
LD 966.01  ; FLOW K2 OK
OR C06_IND_VST80_K2  ; Z
ANDLD
OUT VST80_K2_HJ17
LD TR0
AND K2_TR15_TID_S  ; KURS 2 TRINN 15 TID
AND VST80_K2_HJ17
AND K2_V_DRIFT_OK
@AND P_1s
LD TR0
LD K2_FASEF_OFFIMP  ; FERDIG-OFF-IMPULS.
OR K2_VMFAS_RESET
@OR VST80_K2_START  ; Z
ANDLD
CNT 0216 VST80_K2_TID_TR16  ; KURS 2 TRINN 16 TID
LD TR0
AND K2_TR15_TID_S  ; KURS 2 TRINN 15 TID
ANDNOT K2_TR16_TID_S  ; KURS 2 TRINN 16 TID
BIN(023) C216 D8794
; rung 22: K2-TRINN17  INTOUCH SIER TRINN 14 LUT LUFTDREN 2 ELLER TRINN 24 DESINFEKT LUFTDREN 2
LD P_On
OUT TR0
AND K2_TR16_TID_S  ; KURS 2 TRINN 16 TID
AND K2_V_DRIFT_OK
ANDNOT K2_FASEFORLENG
@LD P_1s
LD 2403.06  ; STOPP LUFTBLAASING KURS 2
@AND P_0_02s
ORLD
ANDLD
LD TR0
LD K2_FASEF_OFFIMP  ; FERDIG-OFF-IMPULS.
OR K2_VMFAS_RESET
@OR VST80_K2_START  ; Z
ANDLD
CNT 0217 VST80_K2_TID_TR17  ; KURS 2 TRINN 17 TID
LD TR0
AND K2_TR16_TID_S  ; KURS 2 TRINN 16 TID
ANDNOT K2_TR17_TID_S  ; KURS 2 TRINN 17 TID
BIN(023) C217 D8794

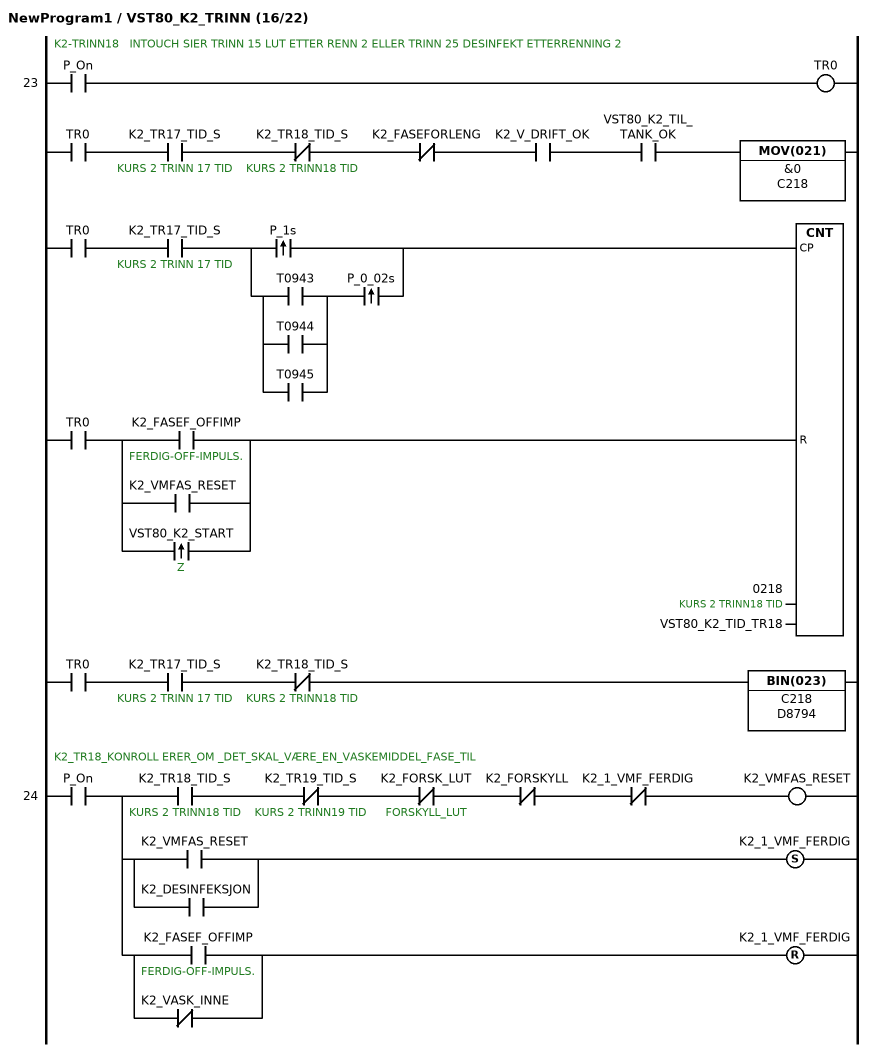
; rung 23: K2-TRINN18   INTOUCH SIER TRINN 15 LUT ETTER RENN 2 ELLER TRINN 25 DESINFEKT ETTERRENNING 2
LD P_On
OUT TR0
AND K2_TR17_TID_S  ; KURS 2 TRINN 17 TID
ANDNOT K2_TR18_TID_S  ; KURS 2 TRINN18 TID
ANDNOT K2_FASEFORLENG
AND K2_V_DRIFT_OK
AND VST80_K2_TIL_TANK_OK
MOV(021) &0 C218
LD TR0
AND K2_TR17_TID_S  ; KURS 2 TRINN 17 TID
@LD P_1s
LD T0943
OR T0944
OR T0945
@AND P_0_02s
ORLD
ANDLD
LD TR0
LD K2_FASEF_OFFIMP  ; FERDIG-OFF-IMPULS.
OR K2_VMFAS_RESET
@OR VST80_K2_START  ; Z
ANDLD
CNT 0218 VST80_K2_TID_TR18  ; KURS 2 TRINN18 TID
LD TR0
AND K2_TR17_TID_S  ; KURS 2 TRINN 17 TID
ANDNOT K2_TR18_TID_S  ; KURS 2 TRINN18 TID
BIN(023) C218 D8794
; rung 24: K2_TR18_KONROLL ERER_OM_DET_SKAL_VÆRE_EN_VASKEMIDDEL_FASE_TIL
LD P_On
OUT TR0
AND K2_TR18_TID_S  ; KURS 2 TRINN18 TID
ANDNOT K2_TR19_TID_S  ; KURS 2 TRINN19 TID
ANDNOT K2_FORSK_LUT  ; FORSKYLL_LUT
ANDNOT K2_FORSKYLL
ANDNOT K2_1_VMF_FERDIG
OUT K2_VMFAS_RESET
LD TR0
LD K2_VMFAS_RESET
OR K2_DESINFEKSJON
ANDLD
SET K2_1_VMF_FERDIG
LD TR0
LD K2_FASEF_OFFIMP  ; FERDIG-OFF-IMPULS.
ORNOT K2_VASK_INNE
ANDLD
RSET K2_1_VMF_FERDIG

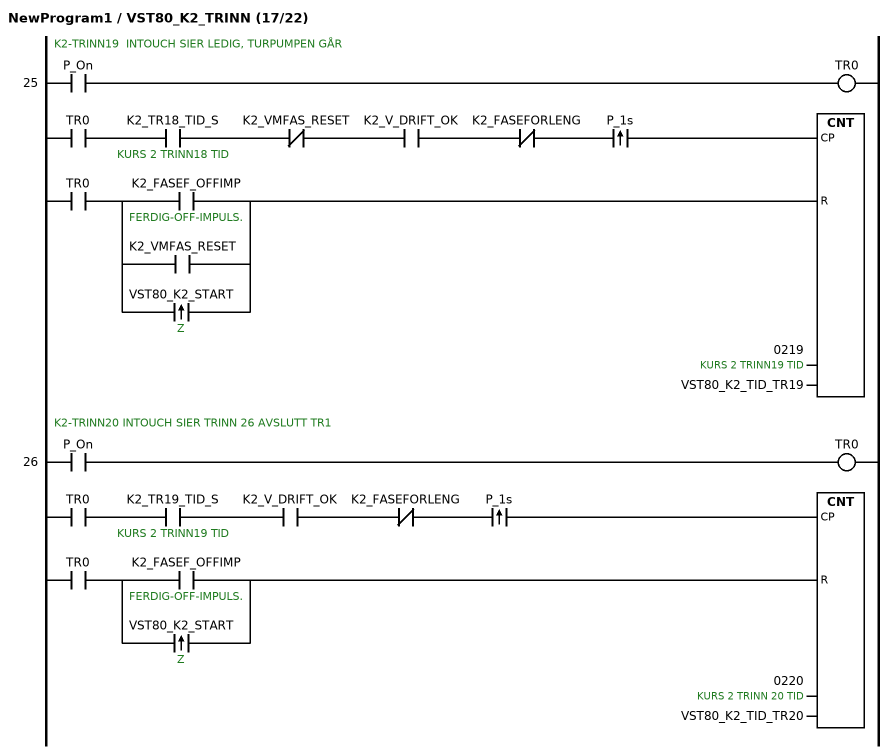
; rung 25: K2-TRINN19  INTOUCH SIER LEDIG, TURPUMPEN GÅR
LD P_On
OUT TR0
AND K2_TR18_TID_S  ; KURS 2 TRINN18 TID
ANDNOT K2_VMFAS_RESET
AND K2_V_DRIFT_OK
ANDNOT K2_FASEFORLENG
@AND P_1s
LD TR0
LD K2_FASEF_OFFIMP  ; FERDIG-OFF-IMPULS.
OR K2_VMFAS_RESET
@OR VST80_K2_START  ; Z
ANDLD
CNT 0219 VST80_K2_TID_TR19  ; KURS 2 TRINN19 TID
; rung 26: K2-TRINN20 INTOUCH SIER TRINN 26 AVSLUTT TR1
LD P_On
OUT TR0
AND K2_TR19_TID_S  ; KURS 2 TRINN19 TID
AND K2_V_DRIFT_OK
ANDNOT K2_FASEFORLENG
@AND P_1s
LD TR0
LD K2_FASEF_OFFIMP  ; FERDIG-OFF-IMPULS.
@OR VST80_K2_START  ; Z
ANDLD
CNT 0220 VST80_K2_TID_TR20  ; KURS 2 TRINN 20 TID

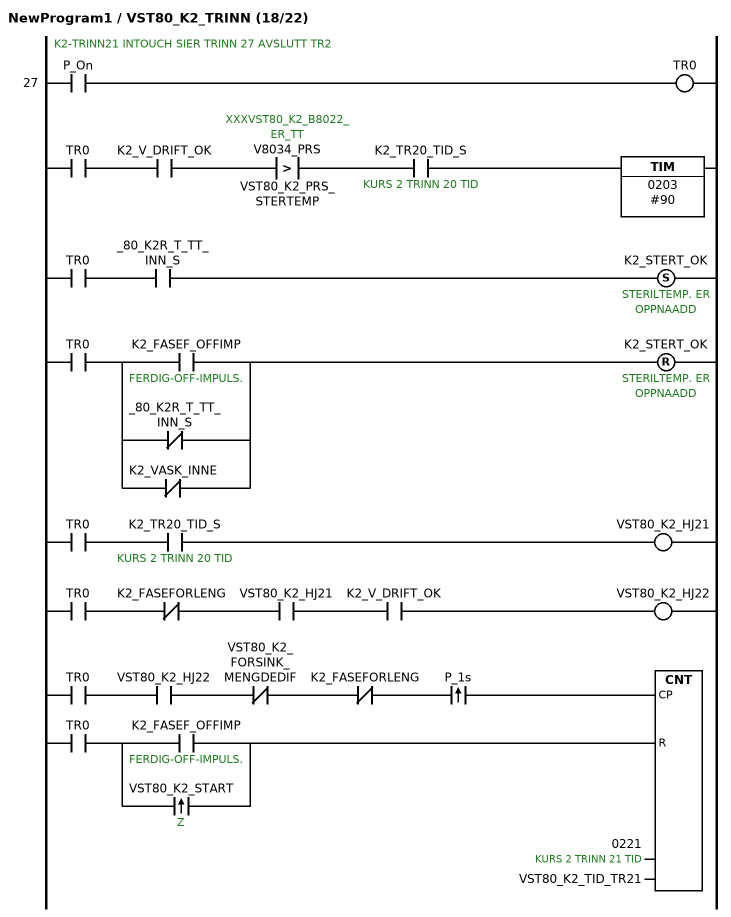
; rung 27: K2-TRINN21 INTOUCH SIER TRINN 27 AVSLUTT TR2
LD P_On
OUT TR0
AND K2_V_DRIFT_OK
AND>(320) V8034_PRS VST80_K2_PRS_STERTEMP  ; XXXVST80_K2_B8022_ER_TT
AND K2_TR20_TID_S  ; KURS 2 TRINN 20 TID
TIM 0203 #90
LD TR0
AND _80_K2R_T_TT_INN_S
SET K2_STERT_OK  ; STERILTEMP. ER OPPNAADD
LD TR0
LD K2_FASEF_OFFIMP  ; FERDIG-OFF-IMPULS.
ORNOT _80_K2R_T_TT_INN_S
ORNOT K2_VASK_INNE
ANDLD
RSET K2_STERT_OK  ; STERILTEMP. ER OPPNAADD
LD TR0
AND K2_TR20_TID_S  ; KURS 2 TRINN 20 TID
OUT VST80_K2_HJ21
LD TR0
ANDNOT K2_FASEFORLENG
AND VST80_K2_HJ21
AND K2_V_DRIFT_OK
OUT VST80_K2_HJ22
LD TR0
AND VST80_K2_HJ22
ANDNOT VST80_K2_FORSINK_MENGDEDIF
ANDNOT K2_FASEFORLENG
@AND P_1s
LD TR0
LD K2_FASEF_OFFIMP  ; FERDIG-OFF-IMPULS.
@OR VST80_K2_START  ; Z
ANDLD
CNT 0221 VST80_K2_TID_TR21  ; KURS 2 TRINN 21 TID

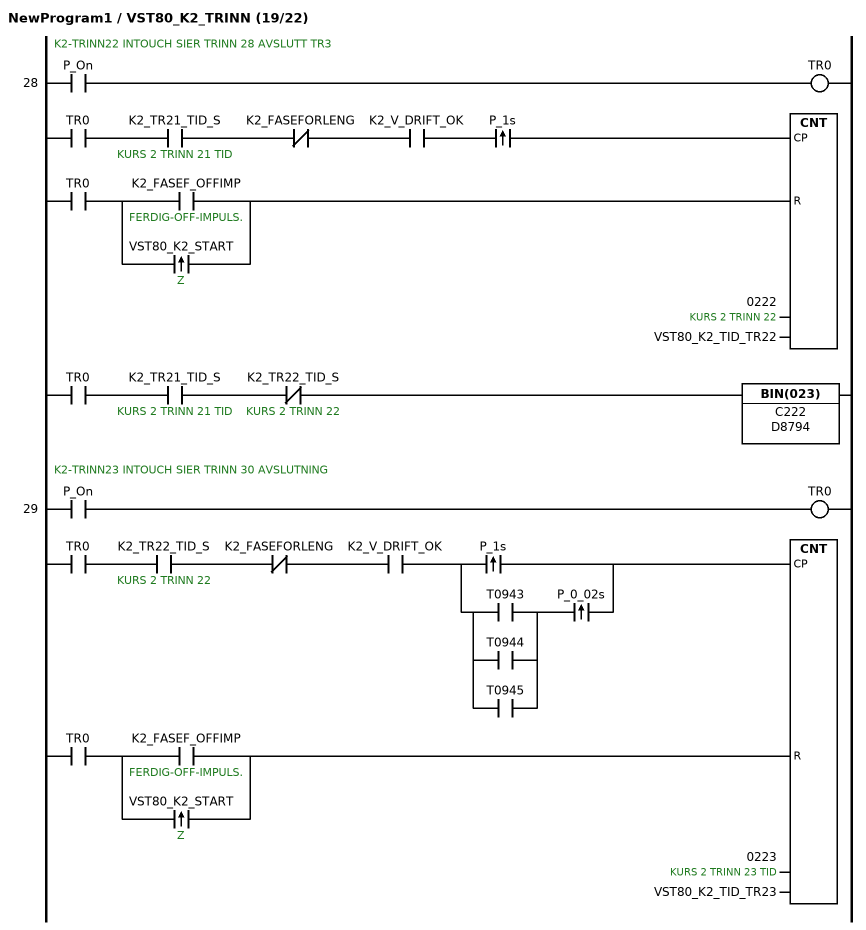
; rung 28: K2-TRINN22 INTOUCH SIER TRINN 28 AVSLUTT TR3
LD P_On
OUT TR0
AND K2_TR21_TID_S  ; KURS 2 TRINN 21 TID
ANDNOT K2_FASEFORLENG
AND K2_V_DRIFT_OK
@AND P_1s
LD TR0
LD K2_FASEF_OFFIMP  ; FERDIG-OFF-IMPULS.
@OR VST80_K2_START  ; Z
ANDLD
CNT 0222 VST80_K2_TID_TR22  ; KURS 2 TRINN 22
LD TR0
AND K2_TR21_TID_S  ; KURS 2 TRINN 21 TID
ANDNOT K2_TR22_TID_S  ; KURS 2 TRINN 22
BIN(023) C222 D8794
; rung 29: K2-TRINN23 INTOUCH SIER TRINN 30 AVSLUTNING
LD P_On
OUT TR0
AND K2_TR22_TID_S  ; KURS 2 TRINN 22
ANDNOT K2_FASEFORLENG
AND K2_V_DRIFT_OK
@LD P_1s
LD T0943
OR T0944
OR T0945
@AND P_0_02s
ORLD
ANDLD
LD TR0
LD K2_FASEF_OFFIMP  ; FERDIG-OFF-IMPULS.
@OR VST80_K2_START  ; Z
ANDLD
CNT 0223 VST80_K2_TID_TR23  ; KURS 2 TRINN 23 TID

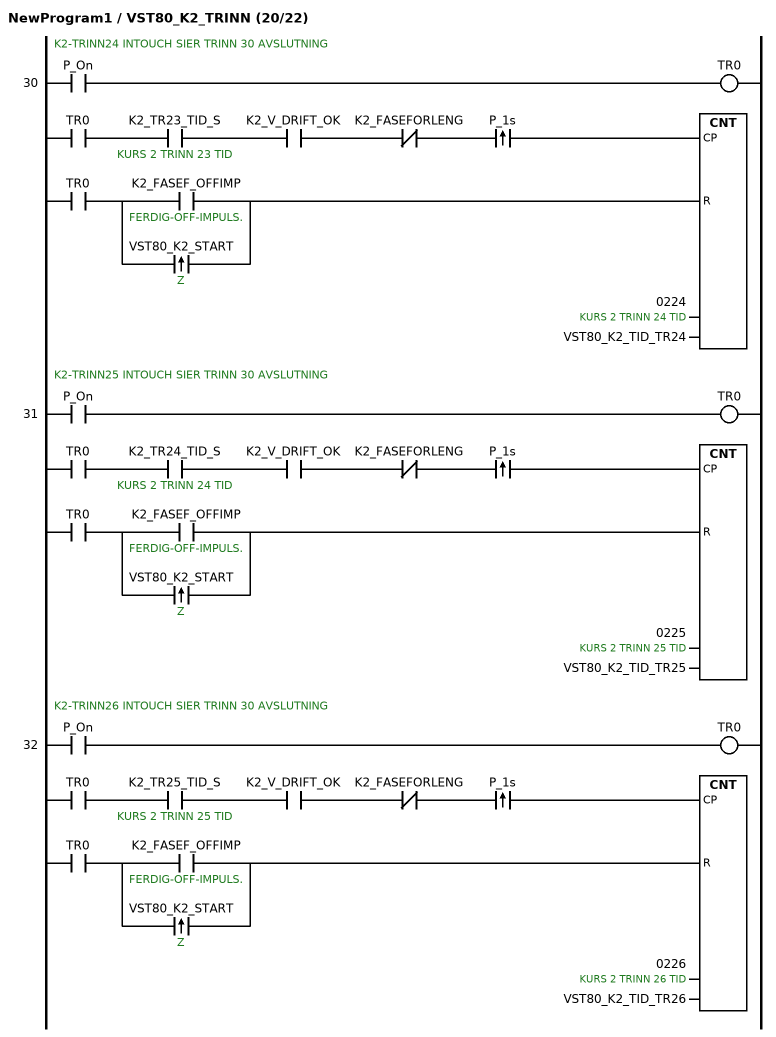
; rung 30: K2-TRINN24 INTOUCH SIER TRINN 30 AVSLUTNING
LD P_On
OUT TR0
AND K2_TR23_TID_S  ; KURS 2 TRINN 23 TID
AND K2_V_DRIFT_OK
ANDNOT K2_FASEFORLENG
@AND P_1s
LD TR0
LD K2_FASEF_OFFIMP  ; FERDIG-OFF-IMPULS.
@OR VST80_K2_START  ; Z
ANDLD
CNT 0224 VST80_K2_TID_TR24  ; KURS 2 TRINN 24 TID
; rung 31: K2-TRINN25 INTOUCH SIER TRINN 30 AVSLUTNING
LD P_On
OUT TR0
AND K2_TR24_TID_S  ; KURS 2 TRINN 24 TID
AND K2_V_DRIFT_OK
ANDNOT K2_FASEFORLENG
@AND P_1s
LD TR0
LD K2_FASEF_OFFIMP  ; FERDIG-OFF-IMPULS.
@OR VST80_K2_START  ; Z
ANDLD
CNT 0225 VST80_K2_TID_TR25  ; KURS 2 TRINN 25 TID
; rung 32: K2-TRINN26 INTOUCH SIER TRINN 30 AVSLUTNING
LD P_On
OUT TR0
AND K2_TR25_TID_S  ; KURS 2 TRINN 25 TID
AND K2_V_DRIFT_OK
ANDNOT K2_FASEFORLENG
@AND P_1s
LD TR0
LD K2_FASEF_OFFIMP  ; FERDIG-OFF-IMPULS.
@OR VST80_K2_START  ; Z
ANDLD
CNT 0226 VST80_K2_TID_TR26  ; KURS 2 TRINN 26 TID

